// TIA Portal project "2022.04.25-PLC上升沿下降沿" (V17)

(* hardware
DEVICE "S7-1500/ET200MP station_1"  S7-1500 station
   slot 0: "导轨_0"  Rack  6ES7 590-1***0-0AA0
   slot 1: "PLC_1"  CPU 1516-3 PN/DP  6ES7 516-3AN00-0AB0  V1.7
      slot 3: "CPU 显示_1"  6ES7591-1BA00-0AA0
      slot 32768: "PROFINET 接口_1"  X1
         slot 32769: "端口_1"  X1 P1
         slot 32770: "端口_2"  X1 P2
      slot 33024: "PROFINET 接口_2"  X2
         slot 33025: "端口_1"  X2 P1
      slot 33280: "DP 接口_1"  X3
   slot 2: "DI 32x24VDC BA_1"  DI 32x24VDC BA  6ES7 521-1BL10-0AA0  V1.1
   slot 3: "DQ 32x24VDC/0.5A HF_1"  DQ 32x24VDC/0.5A HF  6ES7 522-1BL01-0AB0  V1.1
*)

// ===== PLC "PLC_1"  CPU 1516-3 PN/DP =====

VAR_GLOBAL   // PLC tag table "默认变量表"
   "按钮1" AT %I0.0 : Bool;
   "按钮2" AT %I0.1 : Bool;
   "按钮3" AT %I0.2 : Bool;
   "按钮4" AT %I0.3 : Bool;
   "按钮5" AT %I0.4 : Bool;
   "按钮6" AT %I0.5 : Bool;
   "按钮7" AT %I0.6 : Bool;
   "按钮8" AT %I0.7 : Bool;
   "按钮9" AT %I1.0 : Bool;
   "按钮10" AT %I1.1 : Bool;
   "按钮11" AT %I1.2 : Bool;
   "指示灯1" AT %Q0.0 : Bool;
   "指示灯2" AT %Q0.1 : Bool;
   "指示灯3" AT %Q0.2 : Bool;
   "指示灯4" AT %Q0.3 : Bool;
   "指示灯5" AT %Q0.4 : Bool;
   "指示灯6" AT %Q0.5 : Bool;
   "指示灯7" AT %Q0.6 : Bool;
   "指示灯8" AT %Q0.7 : Bool;
   "指示灯9" AT %Q1.0 : Bool;
   "指示灯10" AT %Q1.1 : Bool;
   "指示灯11" AT %Q1.2 : Bool;
   "指示灯12" AT %Q1.3 : Bool;
   "Tag_1" AT %M1.0 : Bool;
   "Tag_2" AT %M1.1 : Bool;
   "Tag_3" AT %M1.2 : Bool;
   "Tag_4" AT %M1.3 : Bool;
   "Tag_5" AT %M1.5 : Bool;
   "Tag_6" AT %M1.6 : Bool;
   "Tag_7" AT %M1.7 : Bool;
   "Tag_8" AT %M2.0 : Bool;
   "Tag_9" AT %M10.0 : Bool;
   "Tag_10" AT %M10.1 : Bool;
   "Tag_11" AT %M10.5 : Bool;
   "Tag_12" AT %M10.6 : Bool;
   "Tag_13" AT %M20.0 : Bool;
   "Tag_14" AT %M20.1 : Bool;
END_VAR

DATA_BLOCK "上升沿下降沿LAD_DB"   // DB1
{ S7_Optimized_Access := 'TRUE' }
VERSION : 0.1
// stored: InstanceOfName 上升沿下降沿LAD
"上升沿下降沿LAD"
BEGIN
END_DATA_BLOCK

DATA_BLOCK "上升下降沿FBD_DB"   // DB4
{ S7_Optimized_Access := 'TRUE' }
VERSION : 0.1
// stored: InstanceOfName 上升下降沿FBD
"上升下降沿FBD"
BEGIN
END_DATA_BLOCK

DATA_BLOCK "上升下降沿SCL_DB"   // DB5
{ S7_Optimized_Access := 'TRUE' }
VERSION : 0.1
// stored: InstanceOfName 上升下降沿SCL
"上升下降沿SCL"
BEGIN
END_DATA_BLOCK

FUNCTION_BLOCK "上升沿下降沿LAD"   // FB1, LAD
{ S7_Optimized_Access := 'TRUE' }
VERSION : 0.1
   VAR_TEMP   // added for the SCL form of the ladder/FBD networks
      _w1 : Bool;
      _w2 : Bool;
   END_VAR
BEGIN

REGION Network 1
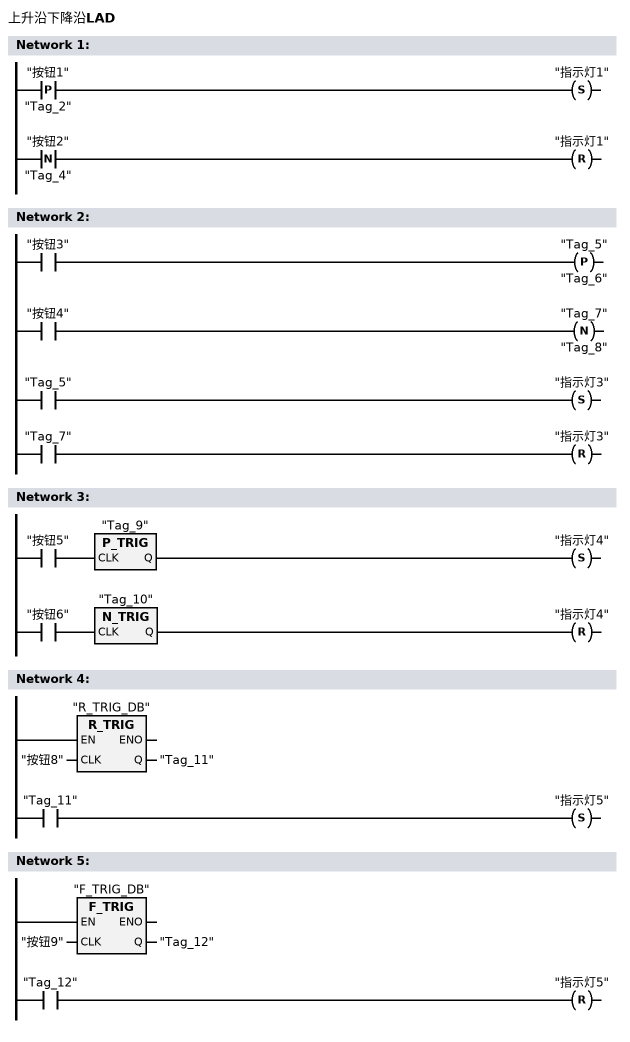
   RUNG wire#powerrail
      P_Contact(operand := "按钮1", bit := "Tag_2")
      S_Coil( "指示灯1" )
   END_RUNG
   RUNG wire#powerrail
      N_Contact(operand := "按钮2", bit := "Tag_4")
      R_Coil( "指示灯1" )
   END_RUNG
   // the same network as SCL:
   #_w1 := "按钮1" AND NOT "Tag_2";   // rising edge of "按钮1"
   "Tag_2" := "按钮1";
   IF #_w1 THEN "指示灯1" := TRUE; END_IF;
   #_w2 := NOT "按钮2" AND "Tag_4";   // falling edge of "按钮2"
   "Tag_4" := "按钮2";
   IF #_w2 THEN "指示灯1" := FALSE; END_IF;
END_REGION

REGION Network 2
   "Tag_5" := "按钮3" AND NOT "Tag_6";   // rising edge
   "Tag_6" := "按钮3";
   "Tag_7" := NOT "按钮4" AND "Tag_8";   // falling edge
   "Tag_8" := "按钮4";
   IF "Tag_5" THEN "指示灯3" := TRUE; END_IF;
   IF "Tag_7" THEN "指示灯3" := FALSE; END_IF;
END_REGION

REGION Network 3
   RUNG wire#powerrail
      Contact( "按钮5" )
      P_Trig( "Tag_9" )
      S_Coil( "指示灯4" )
   END_RUNG
   RUNG wire#powerrail
      Contact( "按钮6" )
      N_Trig( "Tag_10" )
      R_Coil( "指示灯4" )
   END_RUNG
   // the same network as SCL:
   #_w1 := "按钮5" AND NOT "Tag_9";   // rising edge
   "Tag_9" := "按钮5";
   IF #_w1 THEN "指示灯4" := TRUE; END_IF;
   #_w2 := NOT "按钮6" AND "Tag_10";   // falling edge
   "Tag_10" := "按钮6";
   IF #_w2 THEN "指示灯4" := FALSE; END_IF;
END_REGION

REGION Network 4
   "R_TRIG_DB"(CLK := "按钮8", Q => "Tag_11");   // R_TRIG
   IF "Tag_11" THEN "指示灯5" := TRUE; END_IF;
END_REGION

REGION Network 5
   "F_TRIG_DB"(CLK := "按钮9", Q => "Tag_12");   // F_TRIG
   IF "Tag_12" THEN "指示灯5" := FALSE; END_IF;
END_REGION
END_FUNCTION_BLOCK

FUNCTION_BLOCK "上升下降沿FBD"   // FB2, FBD
{ S7_Optimized_Access := 'TRUE' }
VERSION : 0.1
   VAR
      R_TRIG_Instance : R_TRIG;
      F_TRIG_Instance : F_TRIG;
   END_VAR
   VAR_TEMP   // added for the SCL form of the ladder/FBD networks
      _w1 : Bool;
      _w2 : Bool;
   END_VAR
BEGIN

REGION Network 1
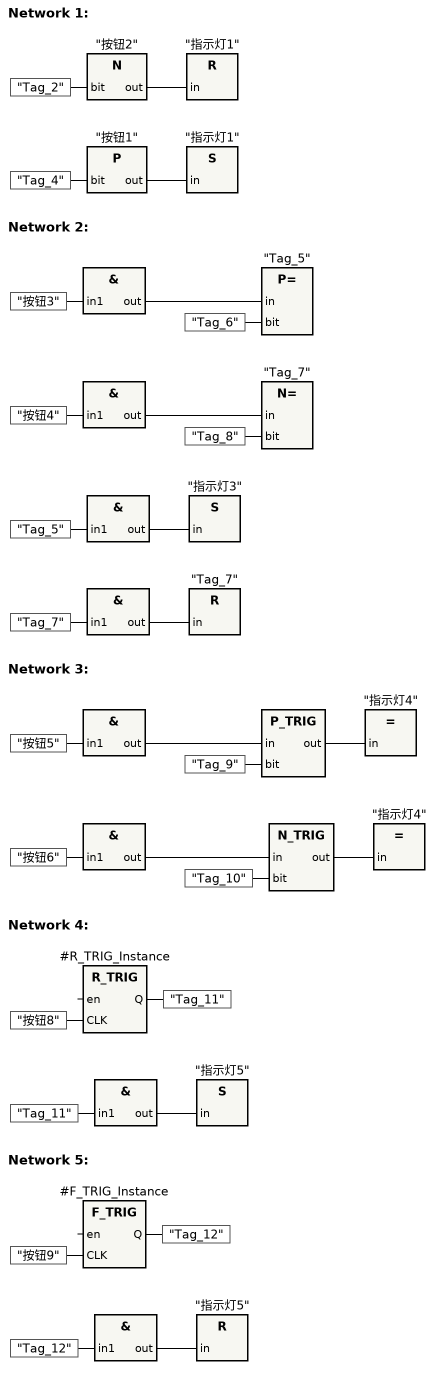
   #_w1 := NOT "按钮2" AND "Tag_2";   // falling edge of "按钮2"
   "Tag_2" := "按钮2";
   IF #_w1 THEN "指示灯1" := FALSE; END_IF;
   #_w2 := "按钮1" AND NOT "Tag_4";   // rising edge of "按钮1"
   "Tag_4" := "按钮1";
   IF #_w2 THEN "指示灯1" := TRUE; END_IF;
END_REGION

REGION Network 2
   "Tag_5" := "按钮3" AND NOT "Tag_6";   // rising edge
   "Tag_6" := "按钮3";
   "Tag_7" := NOT "按钮4" AND "Tag_8";   // falling edge
   "Tag_8" := "按钮4";
   IF "Tag_5" THEN "指示灯3" := TRUE; END_IF;
   IF "Tag_7" THEN "Tag_7" := FALSE; END_IF;
END_REGION

REGION Network 3
   #_w1 := "按钮5" AND NOT "Tag_9";   // rising edge
   "Tag_9" := "按钮5";
   "指示灯4" := #_w1;
   #_w2 := NOT "按钮6" AND "Tag_10";   // falling edge
   "Tag_10" := "按钮6";
   "指示灯4" := #_w2;
END_REGION

REGION Network 4
   #R_TRIG_Instance(CLK := "按钮8", Q => "Tag_11");   // R_TRIG
   IF "Tag_11" THEN "指示灯5" := TRUE; END_IF;
END_REGION

REGION Network 5
   #F_TRIG_Instance(CLK := "按钮9", Q => "Tag_12");   // F_TRIG
   IF "Tag_12" THEN "指示灯5" := FALSE; END_IF;
END_REGION
END_FUNCTION_BLOCK

FUNCTION_BLOCK "上升下降沿SCL"   // FB3, SCL
{ S7_Optimized_Access := 'TRUE' }
VERSION : 0.1
   VAR
      R_TRIG_Instance : R_TRIG;
      F_TRIG_Instance : F_TRIG;
   END_VAR
BEGIN
   #R_TRIG_Instance(CLK:="按钮9",
                    Q=>"Tag_13");
   IF "Tag_13" THEN
       "指示灯10" := 1;
   END_IF;
   #F_TRIG_Instance(CLK :="按钮10",
                    Q => "Tag_14");
   IF "Tag_13" THEN
       "指示灯10" := 0;
   END_IF;
END_FUNCTION_BLOCK

ORGANIZATION_BLOCK "Main"   // OB1, LAD, ProgramCycle
TITLE = "Main Program Sweep (Cycle)"
{ S7_Optimized_Access := 'TRUE' }
VERSION : 0.1
   VAR_INPUT
      Initial_Call : Bool;   // Initial call of this OB
      Remanence : Bool;   // =True, if remanent data are available
   END_VAR
BEGIN

REGION Network 1
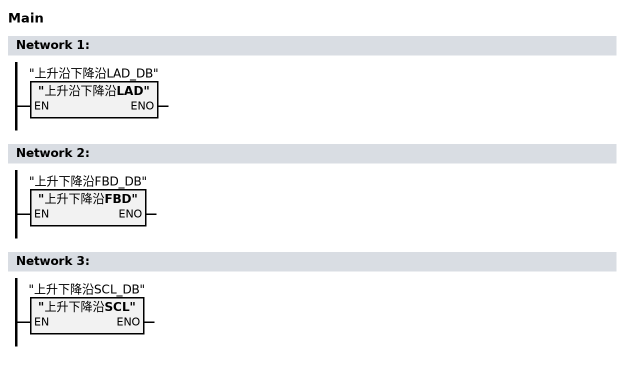
   RUNG wire#powerrail
      "上升沿下降沿LAD_DB"()
   END_RUNG
   // the same network as SCL:
   "上升沿下降沿LAD_DB"();   // "上升沿下降沿LAD"
END_REGION

REGION Network 2
   RUNG wire#powerrail
      "上升下降沿FBD_DB"()
   END_RUNG
   // the same network as SCL:
   "上升下降沿FBD_DB"();   // "上升下降沿FBD"
END_REGION

REGION Network 3
   RUNG wire#powerrail
      "上升下降沿SCL_DB"()
   END_RUNG
   // the same network as SCL:
   "上升下降沿SCL_DB"();   // "上升下降沿SCL"
END_REGION
END_ORGANIZATION_BLOCK